FUNCTION_BLOCK CL_MasterRootClass_old
VAR
  //_nThisIrrLine is either the GHSpan or the Irrigation line.  The irrigation line is some installation coincides with the GHSpan, in other installation is one of the 2 lines of the GHSpan
  //_nThisIrrLine               : UINT :=0; //contain the irrigation line = irrigation line array index to which the object refer to
  //_nThisIrrLineFixedID        : UINT :=0; //contain the irrigation line FixedID derived from EL008 harware bit selector
  
  _IrrLine                    : ST_LineReference;
  
  i01                         : INT := 0;
  nHistoryStep_AR01           : ARRAY[0..C.uiHistoStep_C] OF INT;
  nLastStep01                 : INT := -1;
  
  i02                         : INT := 0;
  nHistoryStep_AR02           : ARRAY[0..C.uiHistoStep_C] OF INT;
  nLastStep02                 : INT := -1;
  
  i03                         : INT := 0;
  nHistoryStep_AR03           : ARRAY[0..C.uiHistoStep_C] OF INT;
  nLastStep03                 : INT := -1;
END_VAR

METHOD Case01Hysto : BOOL
VAR_INPUT
	nStep : INT;
END_VAR
IF nStep <> nLastStep01 THEN
  nLastStep01 := nStep;
  nHistoryStep_AR01[i01] := nStep;
  i01 := i01 + 1;
  IF i01 > C.uiHistoStep_C THEN
    i01 := 0;
  END_IF
END_IF
END_METHOD

METHOD Case01HystoRev : BOOL
VAR_INPUT
	nStep : INT;
END_VAR
IF nStep <> nLastStep01 THEN
  nLastStep01 := nStep;
  FOR i01:= C.uiHistoStep_C TO 1 BY -1 DO
    nHistoryStep_AR01[i01] := nHistoryStep_AR01[i01-1];
  END_FOR
  nHistoryStep_AR01[0] := nStep;
END_IF
END_METHOD

METHOD Case02Hysto : BOOL
VAR_INPUT
	nStep : INT;
END_VAR
IF nStep <> nLastStep02 THEN
  nLastStep02 := nStep;
  nHistoryStep_AR02[i02] := nStep;
  i02 := i02 + 1;
  IF i02 > C.uiHistoStep_C THEN
    i02 := 0;
  END_IF
END_IF
END_METHOD

METHOD Case02HystoRev : BOOL
VAR_INPUT
	nStep : INT;
END_VAR
IF nStep <> nLastStep02 THEN
  nLastStep02 := nStep;
  FOR i02:= C.uiHistoStep_C TO 1 BY -1 DO
    nHistoryStep_AR02[i02] := nHistoryStep_AR02[i02-1];
  END_FOR
  nHistoryStep_AR02[0] := nStep;
END_IF
END_METHOD

METHOD Case03Hysto : BOOL
VAR_INPUT
	nStep : INT;
END_VAR
IF nStep <> nLastStep03 THEN
  nLastStep03 := nStep;
  nHistoryStep_AR03[i03] := nStep;
  i03 := i03 + 1;
  IF i03 > C.uiHistoStep_C THEN
    i03 := 0;
  END_IF
END_IF
END_METHOD

METHOD Case03HystoRev : BOOL
VAR_INPUT
	nStep : INT;
END_VAR
IF nStep <> nLastStep03 THEN
  nLastStep03 := nStep;
  FOR i03:= C.uiHistoStep_C TO 1 BY -1 DO
    nHistoryStep_AR03[i03] := nHistoryStep_AR03[i03-1];
  END_FOR
  nHistoryStep_AR03[0] := nStep;
END_IF
END_METHOD

METHOD Clear01Hysto : BOOL
VAR_INPUT
	nStep : INT;
END_VAR
FOR i01:= 1 TO C.uiHistoStep_C DO
    nHistoryStep_AR01[i01] := 0;
END_FOR
END_METHOD

METHOD Clear02Hysto : BOOL
VAR_INPUT
	nStep : INT;
END_VAR
FOR i02:= 1 TO C.uiHistoStep_C DO
    nHistoryStep_AR02[i02] := 0;
END_FOR
END_METHOD

METHOD Clear03Hysto : BOOL
VAR_INPUT
	nStep : INT;
END_VAR
FOR i03:= 1 TO C.uiHistoStep_C DO
    nHistoryStep_AR03[i03] := 0;
END_FOR
END_METHOD

PROPERTY PUBLIC MRIrrLine : UINT
GET
MRIrrLine := _IrrLine.nThis;
END_GET
SET
_IrrLine.nThis := MRIrrLine;
END_SET
END_PROPERTY

PROPERTY PUBLIC MRIrrLineFixedID : UINT
GET
MRIrrLineFixedID := _IrrLine.nFixedID;
END_GET
SET
_IrrLine.nFixedID := MRIrrLineFixedID;
END_SET
END_PROPERTY

PROPERTY PUBLIC MRLineRef : ST_LineReference
GET
MRLineRef := _IrrLine;
END_GET
SET
_IrrLine := MRLineRef;
END_SET
END_PROPERTY

END_FUNCTION_BLOCK

(* stored: Version 1.1.0.1, ProductVersion 3.1.4024.13
   POU CL_MasterRootClass_old: Id {92d25d2e-4038-4367-a45e-53b08684dc3c}, SpecialFunc None
   Method Case01Hysto: Id {c21a2dba-35ab-4cc2-91c9-ebd77c3d948b}
   Method Case01HystoRev: Id {05c1cd39-1341-4456-acbf-aaabc40f38ff}
   Method Case02Hysto: Id {a2444fb3-18dd-43f4-b541-ebf6036e4d70}
   Method Case02HystoRev: Id {4221a86b-9ab8-416c-9669-0164f1154473}
   Method Case03Hysto: Id {1ab83e67-a34d-442d-9abc-a21e249fb1a6}
   Method Case03HystoRev: Id {eddf62dc-2e7c-4166-9738-717fe887a6ec}
   Method Clear01Hysto: Id {757feae8-ce88-4503-a180-25caa29299c8}
   Method Clear02Hysto: Id {2ec5d523-bbc8-4d9a-ae4e-d82efd5bfa84}
   Method Clear03Hysto: Id {23c5198b-2248-4d9d-a536-f429a2c3edd2}
   Property MRIrrLine: Id {a62cf50e-0076-49bb-925b-c951f230b89c}
   Get Get: Id {ac628814-c561-4cfd-9afd-12c62979e6ff}
   Set Set: Id {aa2ee292-0fcc-4562-a706-6d95519b76ba}
   Property MRIrrLineFixedID: Id {f073a66a-e12a-4769-83ce-c9de4fb06daa}
   Get Get: Id {f78e31cb-def3-4767-a6a4-f388e148c0b6}
   Set Set: Id {2ccb50ab-cf67-449c-80e5-588f1b5ac48f}
   Property MRLineRef: Id {bac79d96-2606-4306-b34f-d5a6c1117aaa}
   Get Get: Id {8bcc770a-96f5-40e1-9a72-5d56750996a7}
   Set Set: Id {e96f5dba-3745-495f-b046-686eb7fc2f4f} *)
